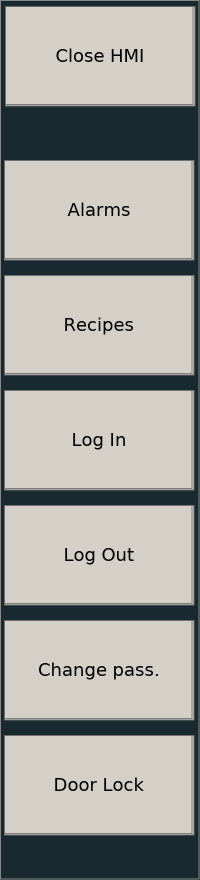
VISUALIZATION NavBarAuxilary_1  // 200x880
VAR_IN_OUT
	btnAlarms			: BOOL;
	btnRecipes			: BOOL;
	btnDoorLock			: BOOL;
	btnLogIn			: BOOL;
	btnLogOut			: BOOL;
	btnHmiClose			: BOOL;
	sCloseHMIFileName	: STRING;
	sCloseHMIParameters	: STRING;
	
	bVisNotInit 		: BOOL;
	bVisHmiCLose		: BOOL;
	bVisLogIn			: BOOL;
	bVisLogOut			: BOOL;
	bDoorLockDisabled	: BOOL;
	bDoorLockInvisible	: BOOL;
END_VAR
    Button (5,6 190x100), "Close HMI", input disabled if: bVisHmiCLose
        tap btnHmiClose
        toggle btnHmiClose
        OnMouseClick: ExecuteCommand ExecuteCommand=ExecuteCommand=[Command=ExecutePlcProgram, Value=sCloseHMIFileName, Value2=sCloseHMIParameters, Command=ExecutePlcProgram]
    Button (4,390 190x100), "Log In", input disabled if: bVisLogIn
        tap btnLogIn
        OnMouseUp: VisuUserMgmt Type=Login
    Button (4,505 190x100), "Log Out", input disabled if: bVisLogOut
        tap btnLogOut
        OnMouseUp: VisuUserMgmt Type=Logout
    Button (4,620 190x100), "Change pass.", input disabled if: bVisLogOut
        OnMouseUp: VisuUserMgmt Type=ChangeUserPassword
    Button (4,160 190x100), "Alarms"
        tap btnAlarms
    Button (4,275 190x100), "Recipes", input disabled if: bVisNotInit
        tap btnRecipes
    Button (4,735 190x100), "Door Lock", invisible if: bDoorLockInvisible, input disabled if: bDoorLockDisabled
        toggle btnDoorLock
END_VISUALIZATION

(* stored: Version 1.1.0.1, ProductVersion 3.1.4024.12
   Visu NavBarAuxilary_1: Id {4dc33e39-ba84-47ca-8b05-210498554a03} *)
